// TIA Portal project "Simulazione" (V16)

(* hardware
DEVICE "S71500/ET200MP station_1"  S7-1500 station
   slot 0: "Telaio di montaggio_0"  Rack  6ES7 590-1***0-0AA0
   slot 1: "PLC_1"  CPU 1512C-1 PN  6ES7 512-1CK01-0AB0  V2.6
      slot 3: "Display CPU_1"  6ES7591-1AA00-0AA0
      slot 32768: "Interfaccia PROFINET_1"  X1
         slot 32769: "Porta_1"  X1 P1
         slot 32770: "Porta_2"  X1 P2
*)

// ===== PLC "PLC_1"  CPU 1512C-1 PN =====

VAR_GLOBAL   // PLC tag table "Tabella delle variabili standard"
   ""Ib1_fisico"" AT %IB1 : Byte;
   ""i1_0_fisico"" AT %I1.0 : Bool;
   ""i1_1_fisico"" AT %I1.1 : Bool;
   ""i1_2_fisico"" AT %I1.2 : Bool;
   ""i1_3_fisico"" AT %I1.3 : Bool;
   ""i1_4_fisico"" AT %I1.4 : Bool;
   ""i1_5_fisico"" AT %I1.5 : Bool;
   ""i1_6_fisico"" AT %I1.6 : Bool;
   ""i1_7_fisico"" AT %I1.7 : Bool;
   ""reset_allarmi_fisico"" AT %I10.3 : Bool;
   ""scelta_fisico"" AT %I10.4 : Bool;
   ""i0_5_fisico"" AT %I10.5 : Bool;
   ""stile_birra_fisico"" AT %I10.0 : Bool;
   ""start_fisico"" AT %I10.1 : Bool;
   ""cip_fisico"" AT %I10.2 : Bool;
   ""i0_6_fisico"" AT %I10.6 : Bool;
   ""abil_fisico"" AT %I10.7 : Bool;
   ""Ib10_fisico"" AT %IB10 : Byte;
   ""livello_analogico"" AT %IW0 : Word;
   ""temperatura_analogico"" AT %IW2 : Word;
   ""pressione_analogico"" AT %IW4 : Word;
   ""QB0"" AT %QB4 : Byte;
   ""ALLARME_ABIL"" AT %Q5.0 : Bool;
   ""ALLARME_LIVELLO"" AT %Q5.1 : Bool;
   ""ALLARME_TEMPERATURA"" AT %Q5.2 : Bool;
   ""ALLARME_PRESSIONE"" AT %Q5.3 : Bool;
   ""V_ACQUA"" AT %Q4.0 : Bool;
   ""V_CARBO"" AT %Q4.4 : Bool;
   ""V_ALCALINA"" AT %Q4.1 : Bool;
   ""V_ACIDO"" AT %Q4.2 : Bool;
   ""V_STERILIZZAZIONE"" AT %Q4.3 : Bool;
   ""V_RAFFREDDAMENTO"" AT %Q4.5 : Bool;
   ""V_TRASF"" AT %Q4.7 : Bool;
   ""QB1"" AT %QB5 : Byte;
   ""ALLARME_SOTTOPRESSIONE"" AT %Q5.4 : Bool;
   ""Q0.6"" AT %Q4.6 : Bool;
END_VAR